// SIMATIC S7-200 project (STEP 7-Micro/WIN), CPU 224 REL 02.01

ORGANIZATION_BLOCK MAIN:OB1
TITLE=PROGRAM COMMENTS
BEGIN
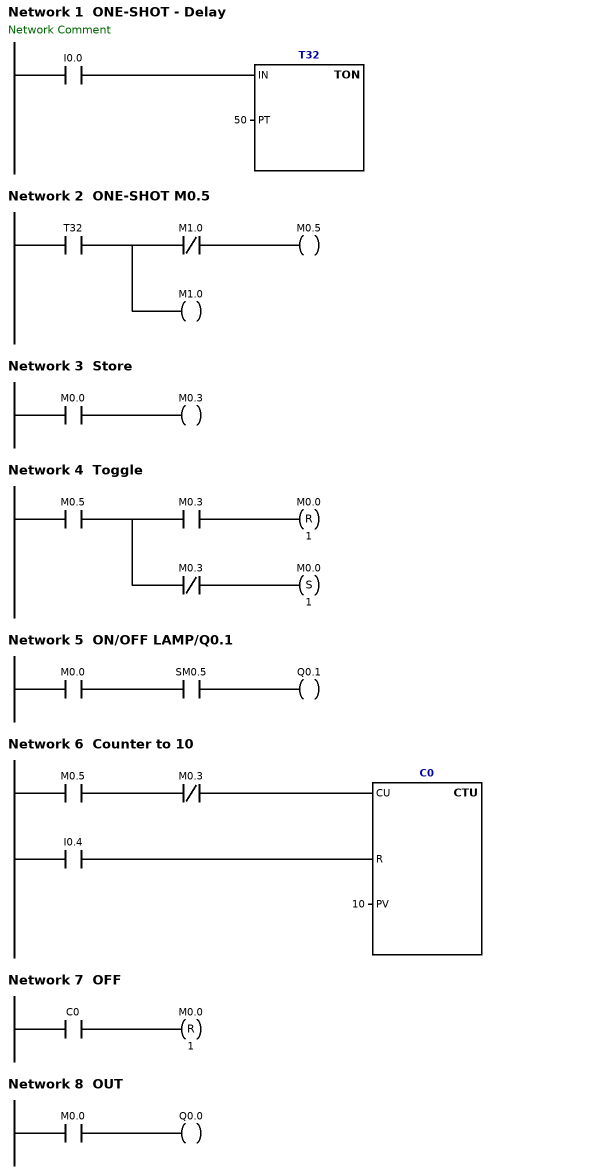
Network 1 // ONE-SHOT - Delay
// Network Comment
LD     I0.0
TON    T32, 50
Network 2 // ONE-SHOT M0.5
LD     T32
LPS
AN     M1.0
=      M0.5
LPP
=      M1.0
Network 3 // Store 
LD     M0.0
=      M0.3
Network 4 // Toggle
LD     M0.5
LPS
A      M0.3
R      M0.0, 1
LPP
AN     M0.3
S      M0.0, 1
Network 5 // ON/OFF LAMP/Q0.1

LD     M0.0
A      SM0.5
=      Q0.1
Network 6 // Counter to 10 
LD     M0.5
AN     M0.3
LD     I0.4
CTU    C0, 10
Network 7 // OFF
LD     C0
R      M0.0, 1
Network 8 // OUT
LD     M0.0
=      Q0.0
END_ORGANIZATION_BLOCK
